FUNCTION F_RTrimEx : T_MaxString // removes n characters from end of string
VAR_INPUT
   n : UINT; 
   str : T_MaxString;
END_VAR
VAR
    Length : UINT;
END_VAR

Length := INT_TO_UINT(LEN(str));
IF n > 0 AND n < Length THEN
    // overwrite chars to be trimmed with nulls...
    MEMSET(destAddr := ADR(str) + Length - n,
           fillByte:= 0,
           n := n); 
    
END_IF
F_RTrimEx := str;

END_FUNCTION

(* stored: Version 1.1.0.1, ProductVersion 3.1.4024.3
   POU F_RTrimEx: Id {c2f1bd2b-d31d-43e4-836e-705c34495475}, SpecialFunc None *)
